Staubli VAL3: anyBool.pgx

public program anyBool(bool& x_bInput[], string x_sBool, bool& x_bResult)
  local num l_nLength
  local num l_nElement
begin

  l_nLength = size(x_bInput)
  x_bResult = false

  for l_nElement = 0 to l_nLength-1
    if x_bInput[l_nElement] == false
      if x_sBool == "false" or x_sBool == "False" or x_sBool == "FALSE"
        x_bResult = true
        return
      elseIf x_sBool == "true" or x_sBool == "True" or x_sBool == "TRUE"
        x_bResult = false
      endIf
    elseIf x_bInput[l_nElement] == true
      if x_sBool == "false" or x_sBool == "False" or x_sBool == "FALSE"
        x_bResult = false
      elseIf x_sBool == "true" or x_sBool == "True" or x_sBool == "TRUE"
        x_bResult = true
        return
      endIf
    endIf
  endFor


end
